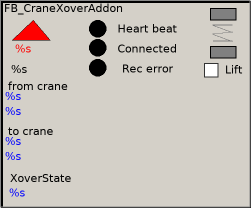
VISUALIZATION V_CraneXoverAddon  // 251x208
VAR_IN_OUT
	{attribute 'VAR_IN_OUT_AS_POINTER'}
	fbFunction		: FB_CraneXoverAddon;	

END_VAR
    Rectangle (1,1 250x207)
    Label (1,1 200x15), "FB_CraneXoverAddon"
    Rectangle (12,39 70x20), "%s", text variable: fbFunction.ZoneData[1].ErrorData.Error.ErrorCode.Conv, invisible if: fbFunction.FunctionData.ErrorData.Error.ErrorCode.Conv = 0
    Polygon (12,40) (33,20) (50,40) (44,40) (22,40), invisible if: fbFunction.FunctionData.ErrorData.ErrorState = E_ErrorState.OPERATIONAL
    Rectangle (6,183 239x20), "%s", tooltip "XoverState", text variable: fbFunction._XoverState
    Rectangle (2,149 248x15), "%s", text variable: fbFunction.HW_Outputs.HandshakeCraneInterfaceSend.HandOverState
    Rectangle (2,134 246x15), "%s", text variable: fbFunction.HW_Outputs.HandshakeCraneInterfaceSend.TakeOverState
    Label (5,124 124x15), "to crane"
    Rectangle (2,89 245x15), "%s", text variable: fbFunction.Inputs.HandshakeCraneInterfaceReceive.TakeOverState
    Rectangle (2,104 246x15), "%s", text variable: fbFunction.Inputs.HandshakeCraneInterfaceReceive.HandOverState
    Label (5,79 124x15), "from crane"
    Rectangle (210,8 26x12), tooltip "Upper lift sensor", colour toggle: fbFunction.HW_Inputs.Sensor_Pos_Up
    Rectangle (210,46 26x12), tooltip "Lower lift sensor", colour toggle: fbFunction.HW_Inputs.Sensor_Pos_Down
    Polyline (232,25) (213,25) (232,32) (213,34) (232,41) (213,41), colour toggle: fbFunction.HW_Outputs.Drive_Run_UpDown
    Label (7,171 124x15), "XoverState"
    Checkbox (202,60 49x20), "Lift", variable: fbFunction.Settings.LiftEnabled, input disabled if: TRUE
    Ellipse (89,20 17x17), colour toggle: fbFunction.HW_Inputs.HandshakeCraneInterfaceReceive.Watchdog
    Label (109,21 77x16), "Heart beat"
    Ellipse (89,39 17x17), colour toggle: fbFunction._fbCranePlcTcpcom.Connected
    Ellipse (89,59 17x17), colour toggle: fbFunction._fbCranePlcTcpcom.ReceiveDataError
    Label (109,41 77x16), "Connected"
    Label (109,61 77x16), "Rec error"
    Rectangle (8,62 76x15), "%s", text variable: fbFunction._fbCranePlcTcpcom.Config.RemotePort
END_VISUALIZATION

(* stored: Version 1.1.0.1, ProductVersion 3.1.4024.9
   Visu V_CraneXoverAddon: Id {68045b8a-0e55-4867-8d73-cf7f657b45c8} *)
